(* IEC 61131-3 sources: CodesysTest/alpha/export/FBs/DataHandlers/ModbusLongHandlerFB.pou, 2 files *)

(* ---- PackDirect.m.st ---- *)
(*#-#-#-#-#-#-#-#-#-#---Declaration---#-#-#-#-#-#-#-#-#-#-#-#-#*)

METHOD PackDirect : ModbusLongType
VAR_INPUT
    highWord : WORD;
    lowWord : WORD
;END_VAR
(*#-#-#-#-#-#-#-#-#-#---Implementation---#-#-#-#-#-#-#-#-#-#-#-#-#*)

PackDirect.rawValue :=  DWORD_TO_DINT(OSCAT_BASIC.DWORD_OF_WORD(highWord,lowWord));

(* ---- Unpack.m.st ---- *)
(*#-#-#-#-#-#-#-#-#-#---Declaration---#-#-#-#-#-#-#-#-#-#-#-#-#*)

METHOD Unpack
VAR_IN_OUT
    modbusLong : ModbusLongType;
END_VAR
(*#-#-#-#-#-#-#-#-#-#---Implementation---#-#-#-#-#-#-#-#-#-#-#-#-#*)

modbusLong.highWord := OSCAT_BASIC.WORD_OF_DWORD(in := DINT_TO_DWORD(modbusLong.rawValue), N := 1);
modbusLong.lowWord := OSCAT_BASIC.WORD_OF_DWORD(in := DINT_TO_DWORD(modbusLong.rawValue), N := 0);
